// LS Electric XG5000 project: 최종 plc 프레임_test
// PLC LSPLC
// module base 0 slot 0: 입출력 모듈:XBC-DR32H (DC 24V 입력, 릴레이 출력 32점)

PROGRAM NewProgram (task: 스캔 프로그램)

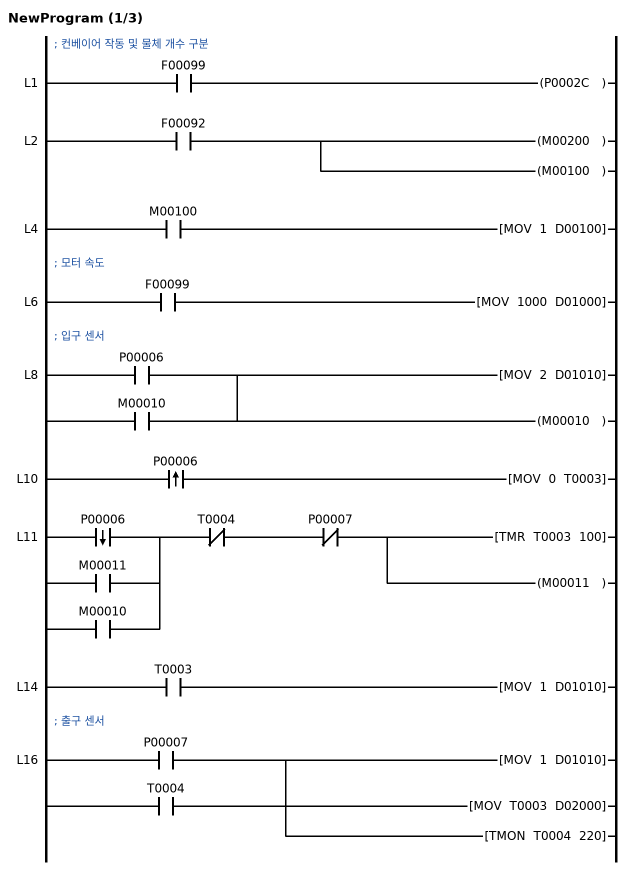
// 컨베이어 작동 및 물체 개수 구분
; L1
LOAD      F00099
OUT       P0002C
; L2
LOAD      F00092
OUT       M00200
OUT       M00100
; L4
LOAD      M00100
MOV       1 D00100
// 모터 속도
; L6
LOAD      F00099
MOV       1000 D01000
// 입구 센서
; L8
LOAD      P00006
OR        M00010
MOV       2 D01010
OUT       M00010
; L10
LOADP     P00006
MOV       0 T0003
; L11
LOADN     P00006
OR        M00011
OR        M00010
AND NOT   T0004
AND NOT   P00007
TMR       T0003 100
OUT       M00011
; L14
LOAD      T0003
MOV       1 D01010
// 출구 센서
; L16
LOAD      P00007
OR        T0004
MOV       1 D01010
MOV       T0003 D02000
TMON      T0004 220

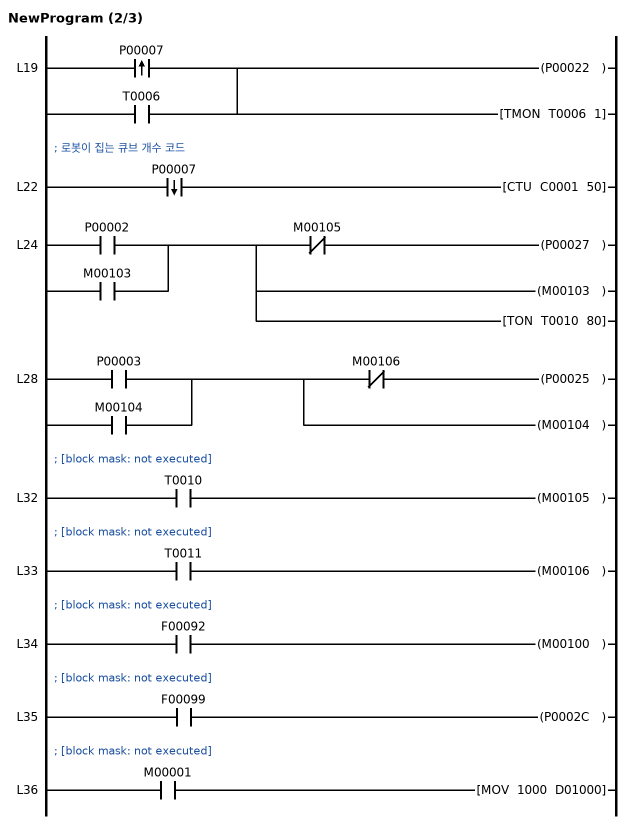
; L19
LOADP     P00007
OR        T0006
OUT       P00022
TMON      T0006 1
// 로봇이 집는 큐브 개수 코드
; L22
LOADN     P00007
CTU       C0001 50
; L24
LOAD      P00002
OR        M00103
MPUSH
AND NOT   M00105
OUT       P00027
MPOP
OUT       M00103
TON       T0010 80
; L28
LOAD      P00003
OR        M00104
MPUSH
AND NOT   M00106
OUT       P00025
MPOP
OUT       M00104
; L32 (block mask: not executed)
LOAD      T0010
OUT       M00105
; L33 (block mask: not executed)
LOAD      T0011
OUT       M00106
; L34 (block mask: not executed)
LOAD      F00092
OUT       M00100
; L35 (block mask: not executed)
LOAD      F00099
OUT       P0002C
; L36 (block mask: not executed)
LOAD      M00001
MOV       1000 D01000

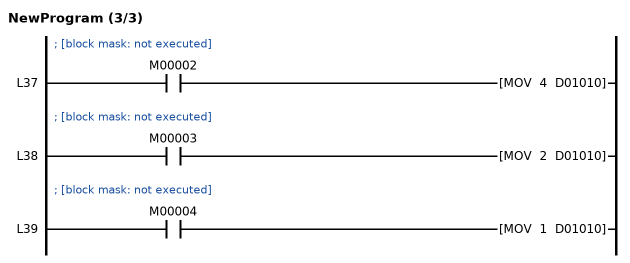
; L37 (block mask: not executed)
LOAD      M00002
MOV       4 D01010
; L38 (block mask: not executed)
LOAD      M00003
MOV       2 D01010
; L39 (block mask: not executed)
LOAD      M00004
MOV       1 D01010